// SIMATIC S7-200 project (STEP 7-Micro/WIN), CPU 222 REL 02.01

ORGANIZATION_BLOCK MAIN:OB1
TITLE=PROGRAM COMMENTS
BEGIN
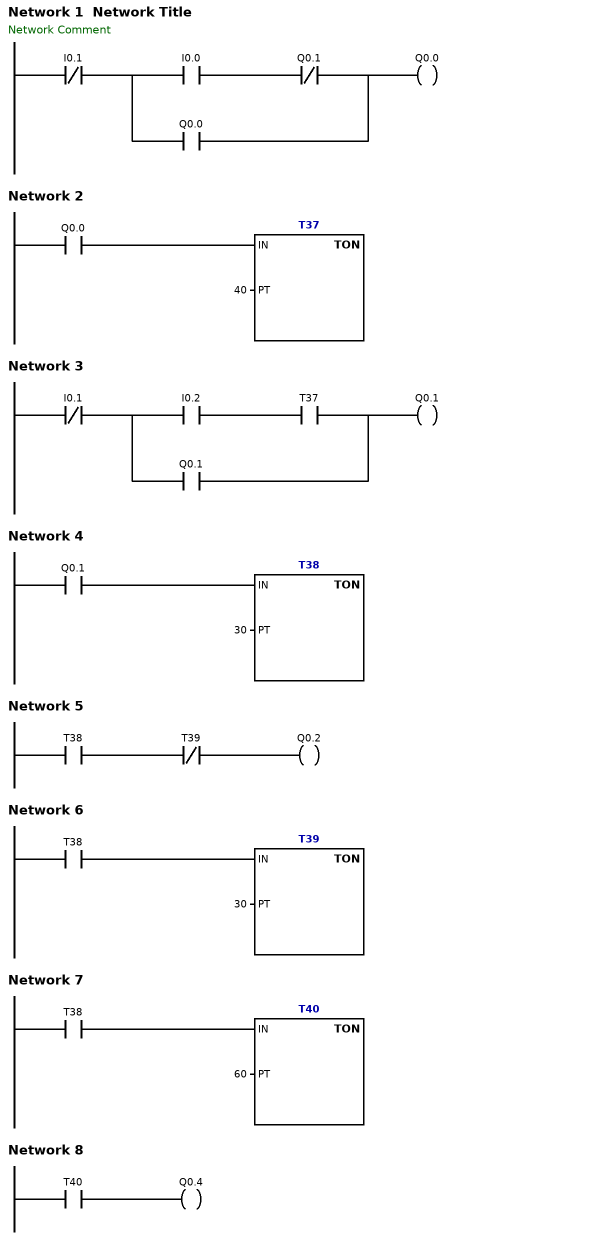
Network 1 // Network Title
// Network Comment
LDN    I0.1
LD     I0.0
AN     Q0.1
O      Q0.0
ALD
=      Q0.0
Network 2
LD     Q0.0
TON    T37, 40
Network 3
LDN    I0.1
LD     I0.2
A      T37
O      Q0.1
ALD
=      Q0.1
Network 4
LD     Q0.1
TON    T38, 30
Network 5
LD     T38
AN     T39
=      Q0.2
Network 6
LD     T38
TON    T39, 30
Network 7
LD     T38
TON    T40, 60
Network 8
LD     T40
=      Q0.4
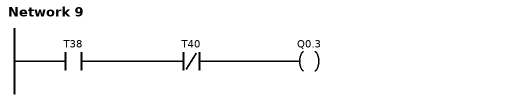
Network 9
LD     T38
AN     T40
=      Q0.3
END_ORGANIZATION_BLOCK
